PROGRAM prgHouse
VAR
	lrHousePower					: LREAL;								//{#lynus.ag#()}

END_VAR

lrHousePower := prgGrid.lrGridPower + prgPv.lrPower_PV1 + prgPv.lrPower_PV2 + prgPv.lrPower_PV3;

END_PROGRAM

(* stored: Version 1.1.0.1, ProductVersion 3.1.4024.12
   POU prgHouse: Id {2627c3a1-fabe-46fd-8396-cc823b8dfb91}, SpecialFunc None *)
